FUNCTION HOUR_TO_TOD : TOD
VAR_INPUT
	IN : REAL;
END_VAR


(*
version 1.2	24. feb 2009
programmer 	hugo
tested by		tobias

converts an amount of hours in real to time of day TOD.

*)

HOUR_TO_TOD := DWORD_TO_TOD(REAL_TO_DWORD(IN * 3600000));


(* revision history
hm	4. aug. 2006	rev 1.0
	original version

hm	14. mar. 2008	rev 1.1
	rounded the input after the last digit

hm	24. feb. 2009	rev 1.2
	changed input to IN
*)

END_FUNCTION

(* stored: Version 1.1.0.1, ProductVersion 3.1.4022.7
   POU HOUR_TO_TOD: Id {c30dd411-20b4-418b-88f6-73d85c94dc12}, SpecialFunc None *)
